Staubli VAL3: GetLimits.pgx

program GetLimits(num& limits[])
begin
  //*******************************************************************************
  //*   ______
  //*  / _____) /|
  //* | |      / /
  //* | | /\  / /
  //* | | \ \/ /  _      Copyright (c) KEOLABS, 2016
  //* | |  \__/  | |        http://www.keolabs.com
  //* | |________| |
  //*  \__________/
  //*
  //********************************************************************************
  //*@file          : GetLimits
  //*@author        : Yves Ragot
  //*@version       : $Id: GetLimits.pgx 1198 2016-10-07 06:48:14Z yves $
  //*@brief         : Get limits
  //*
  //*******************************************************************************/

  // get limits table elements and converts to 1/10 mm
  limits[0] = CurLimitsTable["Xmin"] * 10
  limits[1] = CurLimitsTable["Ymin"] * 10
  limits[2] = CurLimitsTable["Zmin"] * 10
  limits[3] = CurLimitsTable["Xmax"] * 10
  limits[4] = CurLimitsTable["Ymax"] * 10
  limits[5] = CurLimitsTable["Zmax"] * 10

end
